INTERFACE ITF_Group1_HMI_Connector_Command EXTENDS ITF_BaseGroupElement_HMI_Connector_Command

END_INTERFACE

(* stored: Version 1.1.0.1
   Itf ITF_Group1_HMI_Connector_Command: Id {3ed3ea37-3a86-0ab0-1ba3-d7e4696e9ad0} *)
